INTERFACE I_KeyValueCollectionDisposedEvent EXTENDS I_Event

PROPERTY PUBLIC Target : I_KeyValueCollection
GET
END_GET
END_PROPERTY

END_INTERFACE

(* stored: Version 1.1.0.1, ProductVersion 3.1.4024.12
   Itf I_KeyValueCollectionDisposedEvent: Id {3dcb7bae-67a3-0c18-2b5f-903e2567f273}
   Property Target: Id {4b811257-25c6-08bd-1878-e929f4cb7c99}
   Get Get: Id {e46a5376-6daa-09df-180a-1323374e3f36} *)
